FUNCTION_BLOCK FB_Triggers

VAR
	fbRTrig : R_TRIG;
	fbFTrig : F_TRIG;
	bTrigger : BOOL := TRUE;
	bRCount : INT ;
	bFCount : INT ;
	bCycleCount : UDINT ;
END_VAR

fbRTrig( CLK := bTrigger );
fbFTrig (CLK := bTrigger );
IF fbRTrig.Q THEN
	bRCount := bRCount + 1;
END_IF
IF fbFTrig.Q THEN
	bFCount := bFCount + 1;
END_IF
bCycleCount := bCycleCount + 1;

END_FUNCTION_BLOCK

(* stored: Version 1.1.0.1, ProductVersion 3.1.4024.16
   POU FB_Triggers: Id {e08d19c1-115f-4243-816b-1bdb02e9830e}, SpecialFunc None *)
